// TIA Portal V19 export
VAR_GLOBAL   // PLC tag table "D11"
   D11_Lp_EntryReq_LB221 AT %Q108.7 : Bool;   // 232SH1
   D11_Lp_SafetyReset_LB221 AT %Q109.0 : Bool;   // 232SH2
   D11_Pb_EntryReq_LB221 AT %I107.4 : Bool;   // 232SH1
   D11_Pb_SafetyReset_LB221 AT %I107.5 : Bool;   // 232SH2
   D11_Comando_Elettroserratura AT %Q108.6 : Bool;   // 23202
   D11_Cancello_Chiuso AT %I107.2 : Bool;   // 23201
   D11_Cancello_Bloccato AT %I107.3 : Bool;   // 23203
   D11_Ls_Os1 AT %I1072.3 : Bool;   // 105DI3 - 232A1
   D11_Ls_Os2 AT %I1072.7 : Bool;   // 105DI7 - 232A1
END_VAR
